{attribute 'linkalways'} 
{attribute 'no_explicit_call' := 'This FB is a CLASS and must be accessed using methods or properties'}
{attribute 'enable_dynamic_creation'}
FUNCTION_BLOCK FINAL MAX_DWORD EXTENDS Node
VAR
	in1 : _DWORD(0);
	in2 : _DWORD(0);
	out : _DWORD(0);
END_VAR

METHOD PUBLIC Clone : I_Node
VAR
	pNode : POINTER TO MAX_DWORD;
END_VAR
pNode := __NEW(MAX_DWORD);
Clone := pNode^;
END_METHOD

METHOD FB_init : BOOL
VAR_INPUT
	bInitRetains : BOOL; // if TRUE, the retain variables are initialized (warm start / cold start)
	bInCopyCode : BOOL;  // if TRUE, the instance afterwards gets moved into the copy code (online change)
END_VAR
AddInput('in1',THIS^.in1);
AddInput('in2',THIS^.in2);
AddOutput('out', THIS^.out);
END_METHOD

METHOD PROTECTED OnExecute
VAR
END_VAR
out.Value := MAX(in1.Value, in2.Value);
END_METHOD

END_FUNCTION_BLOCK

(* stored: Version 1.1.0.1, ProductVersion 3.1.4024.15
   POU MAX_DWORD: Id {997d57f8-0c1b-427d-a081-aa6c2c89a578}, SpecialFunc None
   Folder Constructor: Id {f713509c-96b3-44a1-bc09-274ee596fa42}
   Method Clone: Id {6dd93ee3-5320-485d-941e-8cccc29f800f}
   Method FB_init: Id {f834535e-c102-4fbf-b23f-37a432bf684c}
   Method OnExecute: Id {6bc4a403-9692-4895-9447-caa035ff8a4b} *)
